(* CoDeSys 2.3.9.45 project: FillingStation.pro *)
(* Libraries: Standard.lib 2.12.10 14:48:34, SYSLIBCALLBACK.LIB 2.12.10 14:48:32 *)

(* PLC configuration (modules and I/O channels)
0753-0553 4 AO 0-20mA [Type_14_4_Channels] node 0, in %IB4 out %QB8 {INTTypePAAssignment = PLC; INTTypeModule = plugged}
  vwPumpPower AT %QW0 [WORDOnW_Q] Ch_1 Analog output
  AT %QW1 [WORDOnW_Q] Ch_2 Analog output
  AT %QW2 [WORDOnW_Q] Ch_3 Analog output
  AT %QW3 [WORDOnW_Q] Ch_4 Analog output
0750-0492 2 AI 4-20mA Diff Measurement Input [Type_8_2_Channels] node 1, in %IB4 out %QB8 {INTTypePAAssignment = PLC; INTTypeModule = plugged}
  vwRawPressure AT %IW0 [WORDOnW_I] Ch_1 Input word
  AT %IW1 [WORDOnW_I] Ch_2 Input word
0750-1515 8 DO 24V DC 0.5A/ 2-wire [Type_10_8_Channels] node 2, in %IB12 out %QB8 {INTTypePAAssignment = PLC; INTTypeModule = plugged}
  vbOpenSamsonValve AT %QX4.0 [BOOLOnX_Q] Ch_1 Digital output
  vbCloseSamsonValve AT %QX4.1 [BOOLOnX_Q] Ch_2 Digital output
  vbOpenDrainValve AT %QX4.2 [BOOLOnX_Q] Ch_3 Digital output
  vbSwitchOnPump AT %QX4.3 [BOOLOnX_Q] Ch_4 Digital output
  AT %QX4.4 [BOOLOnX_Q] Ch_5 Digital output
  AT %QX4.5 [BOOLOnX_Q] Ch_6 Digital output
  AT %QX4.6 [BOOLOnX_Q] Ch_7 Digital output
  AT %QX4.7 [BOOLOnX_Q] Ch_8 Digital output
0750-0459 4 AI 0-10V DC s.e. [Type_8_4_Channels] node 3, in %IB4 out %QB16 {INTTypePAAssignment = PLC; INTTypeModule = plugged}
  vwRawValvePosition AT %IW2 [WORDOnW_I] Ch_1 Input word
  AT %IW3 [WORDOnW_I] Ch_2 Input word
  AT %IW4 [WORDOnW_I] Ch_3 Input word
  AT %IW5 [WORDOnW_I] Ch_4 Input word
Fieldbus variables [FB_VARS] node 1, in %IB0 out %QB0
Flag variables [FLAG_VARS] node 2, in %IB0 out %QB0
Modbus-Master [MB_MASTER] node 3, in %IB0 out %QB0
*)

(* Global variable list: Globale_Variablen *)
VAR_GLOBAL
	vrWaterLevel:REAL;
	vrgrWaterLevel:ARRAY[1..16] OF REAL;
	vrStandardGravity:REAL:=9.81;
	viDensityWater:INT:=1000;
	vrValvePosition:REAL;
	vrValvePositionPercentage:REAL;
	vrValvePositionDesired:REAL;
	viPumpPowerPercentage:INT;
	vbManualValveControl:BOOL:=TRUE;
	vbAutomaticValveControl:BOOL:=FALSE;
	vbPreviousValveControl:STRING:='MANUAL';
	vbPreviousSamsonValveDirection:STRING:='STOP';
	vbStopSamsonValve:BOOL:=TRUE;
END_VAR

(* POU PLC_PRG, FBD *)
PROGRAM PLC_PRG
VAR
END_VAR
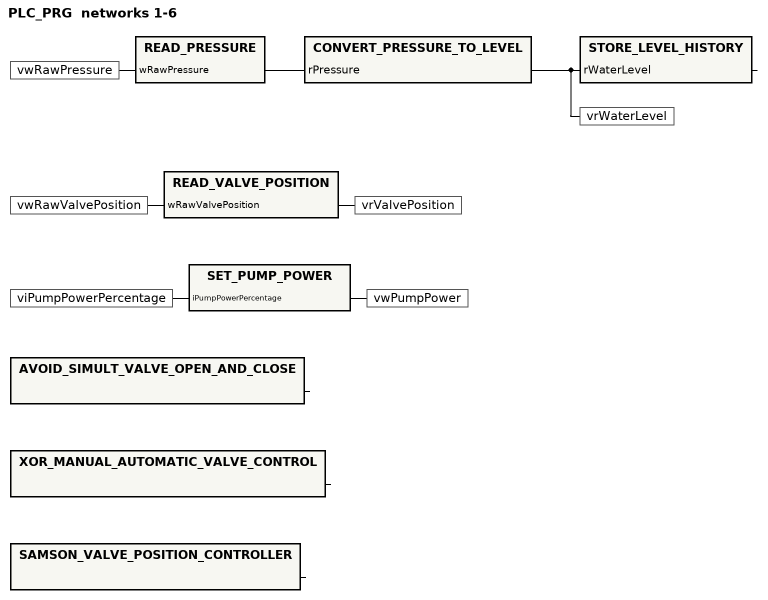
_FBD_ (* Function Block Diagram *)
NETWORK 1
	STORE_LEVEL_HISTORY(rWaterLevel: <CONVERT_PRESSURE_TO_LEVEL(rPressure: READ_PRESSURE(wRawPressure: vwRawPressure)) => vrWaterLevel>)
NETWORK 2
	READ_VALVE_POSITION(wRawValvePosition: vwRawValvePosition) => vrValvePosition
NETWORK 3
	SET_PUMP_POWER(iPumpPowerPercentage: viPumpPowerPercentage) => vwPumpPower
NETWORK 4
	AVOID_SIMULT_VALVE_OPEN_AND_CLOSE()
NETWORK 5
	XOR_MANUAL_AUTOMATIC_VALVE_CONTROL()
NETWORK 6
	SAMSON_VALVE_POSITION_CONTROLLER()
_END_FBD_
(* the same logic as Structured Text *)
(* Network 1: see the listing above *)
(* Network 2 *)
vrValvePosition := READ_VALVE_POSITION(wRawValvePosition := vwRawValvePosition);
(* Network 3 *)
vwPumpPower := SET_PUMP_POWER(iPumpPowerPercentage := viPumpPowerPercentage);
(* Network 4 *)
AVOID_SIMULT_VALVE_OPEN_AND_CLOSE();
(* Network 5 *)
XOR_MANUAL_AUTOMATIC_VALVE_CONTROL();
(* Network 6 *)
SAMSON_VALVE_POSITION_CONTROLLER();
END_PROGRAM

(* POU STORE_LEVEL_HISTORY, ST *)
FUNCTION STORE_LEVEL_HISTORY : BOOL
VAR_INPUT
	rWaterLevel:REAL;
END_VAR
VAR
	index: INT;
	rgrWaterLevelTmp:ARRAY[1..16] OF REAL;
	rgrWaterLevel: REAL;
END_VAR
rgrWaterLevelTmp := vrgrWaterLevel;

FOR index:=1 TO 15 DO
	vrgrWaterLevel[index]:= rgrWaterLevelTmp[index+1];
END_FOR

vrgrWaterLevel[16] := rWaterLevel;
END_FUNCTION

(* POU CONVERT_PRESSURE_TO_LEVEL, ST *)
FUNCTION CONVERT_PRESSURE_TO_LEVEL : REAL
VAR_INPUT
	rPressure:REAL;
END_VAR
VAR
END_VAR
CONVERT_PRESSURE_TO_LEVEL := rPressure/viDensityWater/vrStandardGravity;
END_FUNCTION

(* POU READ_PRESSURE, ST *)
FUNCTION READ_PRESSURE : REAL
VAR_INPUT
	wRawPressure:WORD;
END_VAR
VAR
END_VAR
READ_PRESSURE := WORD_TO_REAL(wRawPressure)/65535*100000;
END_FUNCTION

(* POU READ_VALVE_POSITION, ST *)
FUNCTION READ_VALVE_POSITION : REAL
VAR_INPUT
	wRawValvePosition:WORD;
END_VAR
VAR
END_VAR
READ_VALVE_POSITION := WORD_TO_REAL(wRawValvePosition)/65535*1;
vrValvePositionPercentage := READ_VALVE_POSITION*100;
END_FUNCTION

(* POU SET_PUMP_POWER, ST *)
FUNCTION SET_PUMP_POWER : WORD
VAR_INPUT
	iPumpPowerPercentage: INT;
END_VAR
VAR
END_VAR
SET_PUMP_POWER := INT_TO_WORD(iPumpPowerPercentage)*65535/100;
END_FUNCTION

(* POU AVOID_SIMULT_VALVE_OPEN_AND_CLOSE, ST *)
FUNCTION AVOID_SIMULT_VALVE_OPEN_AND_CLOSE : BOOL
VAR_INPUT
END_VAR
VAR
END_VAR
IF vbOpenSamsonValve AND vbStopSamsonValve THEN
	IF vbPreviousSamsonValveDirection = 'OPEN' THEN
		vbOpenSamsonValve := FALSE;
		vbStopSamsonValve := TRUE;
		vbCloseSamsonValve := FALSE;
		vbPreviousSamsonValveDirection := 'STOP';
	ELSIF vbPreviousSamsonValveDirection = 'STOP' THEN
		vbOpenSamsonValve := TRUE;
		vbStopSamsonValve := FALSE;
		vbCloseSamsonValve := FALSE;
		vbPreviousSamsonValveDirection := 'OPEN';
	END_IF
ELSIF vbStopSamsonValve AND vbCloseSamsonValve THEN
	IF vbPreviousSamsonValveDirection = 'STOP' THEN
		vbOpenSamsonValve := FALSE;
		vbStopSamsonValve := FALSE;
		vbCloseSamsonValve := TRUE;
		vbPreviousSamsonValveDirection := 'CLOSE';
	ELSIF vbPreviousSamsonValveDirection = 'CLOSE' THEN
		vbOpenSamsonValve := FALSE;
		vbStopSamsonValve := TRUE;
		vbCloseSamsonValve := FALSE;
		vbPreviousSamsonValveDirection := 'STOP';
	END_IF
ELSIF vbOpenSamsonValve AND vbCloseSamsonValve THEN
	IF vbPreviousSamsonValveDirection = 'OPEN' THEN
		vbOpenSamsonValve := FALSE;
		vbStopSamsonValve := FALSE;
		vbCloseSamsonValve := TRUE;
		vbPreviousSamsonValveDirection := 'CLOSE';
	ELSIF vbPreviousSamsonValveDirection = 'CLOSE' THEN
		vbOpenSamsonValve := TRUE;
		vbStopSamsonValve := FALSE;
		vbCloseSamsonValve := FALSE;
		vbPreviousSamsonValveDirection := 'OPEN';
	END_IF
END_IF

AVOID_SIMULT_VALVE_OPEN_AND_CLOSE := TRUE;
END_FUNCTION

(* POU XOR_MANUAL_AUTOMATIC_VALVE_CONTROL, ST *)
FUNCTION XOR_MANUAL_AUTOMATIC_VALVE_CONTROL : BOOL
VAR_INPUT
END_VAR
VAR
END_VAR
IF vbAutomaticValveControl AND vbManualValveControl THEN
	IF vbPreviousValveControl = 'MANUAL' THEN
			vbAutomaticValveControl := TRUE;
			vbManualValveControl := FALSE;
			vbPreviousValveControl := 'AUTOMATIC';
	ELSIF
			vbPreviousValveControl =  'AUTOMATIC' THEN
			vbAutomaticValveControl := FALSE;
			vbManualValveControl := TRUE;
			vbPreviousValveControl := 'MANUAL';
	END_IF
END_IF

XOR_MANUAL_AUTOMATIC_VALVE_CONTROL := TRUE;
END_FUNCTION

(* POU SAMSON_VALVE_POSITION_CONTROLLER, ST *)
FUNCTION SAMSON_VALVE_POSITION_CONTROLLER : BOOL
VAR_INPUT
END_VAR
VAR
	delta:REAL:=0.1;
END_VAR
IF vbAutomaticValveControl = TRUE THEN
	IF vrValvePosition < vrValvePositionDesired/100 - delta THEN
		vbOpenSamsonValve := TRUE;
		vbSTOPSamsonValve := FALSE;
		vbCloseSamsonValve := FALSE;
	ELSIF vrValvePosition > vrValvePositionDesired/100 + delta THEN
		vbOpenSamsonValve := FALSE;
		vbSTOPSamsonValve := FALSE;
		vbCloseSamsonValve := TRUE;
	END_IF
END_IF

SAMSON_VALVE_POSITION_CONTROLLER := TRUE;
END_FUNCTION

(* POU Configuration/MODBUS_CONFIGURATION, ST *)
PROGRAM MODBUS_CONFIGURATION        
VAR                                
END_VAR                            
(*                                 
   <?xml version="1.0" encoding="UTF-16" standalone="yes"?>
<network xml_structure_version="1" xml_feature_version="1">
	<generator_settings minRTUTaskCycleTimeMs="5" minEthaskCycleTimeMs="5" ethSlaveMultiplier="0.1" rtuInterfaceMultiplier="0.1" taskGeneration="false"/>
</network>
                              
*)                                 
;                                  
END_PROGRAM

(* Visualisation Filling_Station
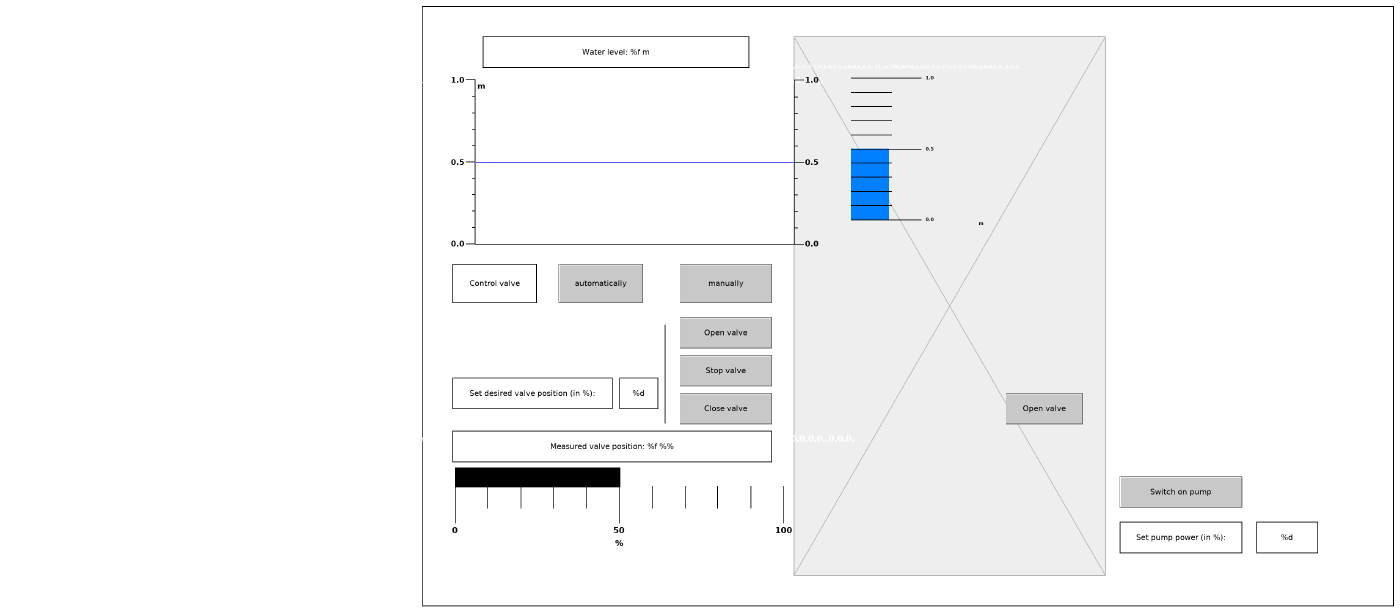
bitmap at (510,60)-(921,771): hydraulics-schematic-simplified.bmp
group at (510,100)-(931,311)
  rectangle at (0,0)-(1,1): text "{ExtendedElement},Visu\ElementDLL.ete,1,@Bargraph,211,421,2,1,0,vrWaterLevel,m,%.1f,0.1,0.5,0,1,0,0,0,0,0,0,0,-13,16,700,Arial,0,128,255,255,0,0,1,100,0,0,0,0,0,,0,0,0,"
  rectangle at (35,203)-(58,379): alarm colour if (vrWaterLevel) > 100; top ((vrWaterLevel * 1.0) - 0.5)  * -352
  rectangle at (80,368)-(196,389): text "0.0"
  rectangle at (80,193)-(196,214): text "0.5"
  rectangle at (80,17)-(196,38): text "1.0"
  rectangle at (103,380)-(127,396): text "m"
group at (60,110)-(541,341)
  rectangle at (0,8)-(1,9): text "{ExtendedElement},Visu\ElementDLL.ete,2,@Histogramm,481,231,vrgrWaterLevel,m,%.1f,0.1,0.5,0,1,0,0,0,0,0,0,0,-13,16,700,Arial,0,0,255,255,0,0,0,0,0,2,1,0_16,0,1,0,,"
  rectangle at (0,231)-(18,247): text "0.0"
  rectangle at (463,231)-(481,247): text "0.0"
  rectangle at (0,116)-(18,132): text "0.5"
  rectangle at (463,116)-(481,132): text "0.5"
  rectangle at (0,0)-(18,16): text "1.0"
  rectangle at (463,0)-(481,16): text "1.0"
  rectangle at (32,8)-(44,25): text "m"
  shape at (31,124)-(57,124): alarm colour if vrgrWaterLevel[0] < 0; top (-1.0 *  vrgrWaterLevel[1]  +  0.5  ) * 231 + SEL( vrgrWaterLevel[1] > 0.5 , 0.5, -0.5); bottom (-1.0 *  vrgrWaterLevel[0]  +  0.5  ) * 231 + SEL( vrgrWaterLevel[0] > 0.5 , 0.5, -0.5)
  shape at (57,124)-(83,124): alarm colour if vrgrWaterLevel[1] < 0; top (-1.0 *  vrgrWaterLevel[2]  +  0.5  ) * 231 + SEL( vrgrWaterLevel[2] > 0.5 , 0.5, -0.5); bottom (-1.0 *  vrgrWaterLevel[1]  +  0.5  ) * 231 + SEL( vrgrWaterLevel[1] > 0.5 , 0.5, -0.5)
  shape at (83,124)-(109,124): alarm colour if vrgrWaterLevel[2] < 0; top (-1.0 *  vrgrWaterLevel[3]  +  0.5  ) * 231 + SEL( vrgrWaterLevel[3] > 0.5 , 0.5, -0.5); bottom (-1.0 *  vrgrWaterLevel[2]  +  0.5  ) * 231 + SEL( vrgrWaterLevel[2] > 0.5 , 0.5, -0.5)
  shape at (109,124)-(135,124): alarm colour if vrgrWaterLevel[3] < 0; top (-1.0 *  vrgrWaterLevel[4]  +  0.5  ) * 231 + SEL( vrgrWaterLevel[4] > 0.5 , 0.5, -0.5); bottom (-1.0 *  vrgrWaterLevel[3]  +  0.5  ) * 231 + SEL( vrgrWaterLevel[3] > 0.5 , 0.5, -0.5)
  shape at (135,124)-(162,124): alarm colour if vrgrWaterLevel[4] < 0; top (-1.0 *  vrgrWaterLevel[5]  +  0.5  ) * 231 + SEL( vrgrWaterLevel[5] > 0.5 , 0.5, -0.5); bottom (-1.0 *  vrgrWaterLevel[4]  +  0.5  ) * 231 + SEL( vrgrWaterLevel[4] > 0.5 , 0.5, -0.5)
  shape at (162,124)-(188,124): alarm colour if vrgrWaterLevel[5] < 0; top (-1.0 *  vrgrWaterLevel[6]  +  0.5  ) * 231 + SEL( vrgrWaterLevel[6] > 0.5 , 0.5, -0.5); bottom (-1.0 *  vrgrWaterLevel[5]  +  0.5  ) * 231 + SEL( vrgrWaterLevel[5] > 0.5 , 0.5, -0.5)
  shape at (188,124)-(214,124): alarm colour if vrgrWaterLevel[6] < 0; top (-1.0 *  vrgrWaterLevel[7]  +  0.5  ) * 231 + SEL( vrgrWaterLevel[7] > 0.5 , 0.5, -0.5); bottom (-1.0 *  vrgrWaterLevel[6]  +  0.5  ) * 231 + SEL( vrgrWaterLevel[6] > 0.5 , 0.5, -0.5)
  shape at (214,124)-(240,124): alarm colour if vrgrWaterLevel[7] < 0; top (-1.0 *  vrgrWaterLevel[8]  +  0.5  ) * 231 + SEL( vrgrWaterLevel[8] > 0.5 , 0.5, -0.5); bottom (-1.0 *  vrgrWaterLevel[7]  +  0.5  ) * 231 + SEL( vrgrWaterLevel[7] > 0.5 , 0.5, -0.5)
  shape at (240,124)-(267,124): alarm colour if vrgrWaterLevel[8] < 0; top (-1.0 *  vrgrWaterLevel[9]  +  0.5  ) * 231 + SEL( vrgrWaterLevel[9] > 0.5 , 0.5, -0.5); bottom (-1.0 *  vrgrWaterLevel[8]  +  0.5  ) * 231 + SEL( vrgrWaterLevel[8] > 0.5 , 0.5, -0.5)
  shape at (267,124)-(293,124): alarm colour if vrgrWaterLevel[9] < 0; top (-1.0 *  vrgrWaterLevel[10]  +  0.5  ) * 231 + SEL( vrgrWaterLevel[10] > 0.5 , 0.5, -0.5); bottom (-1.0 *  vrgrWaterLevel[9]  +  0.5  ) * 231 + SEL( vrgrWaterLevel[9] > 0.5 , 0.5, -0.5)
  shape at (293,124)-(319,124): alarm colour if vrgrWaterLevel[10] < 0; top (-1.0 *  vrgrWaterLevel[11]  +  0.5  ) * 231 + SEL( vrgrWaterLevel[11] > 0.5 , 0.5, -0.5); bottom (-1.0 *  vrgrWaterLevel[10]  +  0.5  ) * 231 + SEL( vrgrWaterLevel[10] > 0.5 , 0.5, -0.5)
  shape at (319,124)-(345,124): alarm colour if vrgrWaterLevel[11] < 0; top (-1.0 *  vrgrWaterLevel[12]  +  0.5  ) * 231 + SEL( vrgrWaterLevel[12] > 0.5 , 0.5, -0.5); bottom (-1.0 *  vrgrWaterLevel[11]  +  0.5  ) * 231 + SEL( vrgrWaterLevel[11] > 0.5 , 0.5, -0.5)
  shape at (345,124)-(372,124): alarm colour if vrgrWaterLevel[12] < 0; top (-1.0 *  vrgrWaterLevel[13]  +  0.5  ) * 231 + SEL( vrgrWaterLevel[13] > 0.5 , 0.5, -0.5); bottom (-1.0 *  vrgrWaterLevel[12]  +  0.5  ) * 231 + SEL( vrgrWaterLevel[12] > 0.5 , 0.5, -0.5)
  shape at (372,124)-(398,124): alarm colour if vrgrWaterLevel[13] < 0; top (-1.0 *  vrgrWaterLevel[14]  +  0.5  ) * 231 + SEL( vrgrWaterLevel[14] > 0.5 , 0.5, -0.5); bottom (-1.0 *  vrgrWaterLevel[13]  +  0.5  ) * 231 + SEL( vrgrWaterLevel[13] > 0.5 , 0.5, -0.5)
  shape at (398,124)-(424,124): alarm colour if vrgrWaterLevel[14] < 0; top (-1.0 *  vrgrWaterLevel[15]  +  0.5  ) * 231 + SEL( vrgrWaterLevel[15] > 0.5 , 0.5, -0.5); bottom (-1.0 *  vrgrWaterLevel[14]  +  0.5  ) * 231 + SEL( vrgrWaterLevel[14] > 0.5 , 0.5, -0.5)
  shape at (424,124)-(450,124): alarm colour if vrgrWaterLevel[15] < 0; top (-1.0 *  vrgrWaterLevel[16]  +  0.5  ) * 231 + SEL( vrgrWaterLevel[16] > 0.5 , 0.5, -0.5); bottom (-1.0 *  vrgrWaterLevel[15]  +  0.5  ) * 231 + SEL( vrgrWaterLevel[15] > 0.5 , 0.5, -0.5)
group at (30,590)-(511,811)
  rectangle at (0,0)-(1,1): text "{ExtendedElement},Visu\ElementDLL.ete,1,@Bargraph,481,221,0,0,0,vrValvePositionPercentage,%,%.0f,10,50,0,100,0,0,0,0,0,0,0,-13,16,700,Arial,0,0,0,255,0,0,0,0,0,0,0,0,0,,0,0,0,"
  rectangle at (32,36)-(241,60): alarm colour if (vrValvePositionPercentage) < 0; right ((vrValvePositionPercentage * 1.0) - 50)  * 4.16
  rectangle at (27,106)-(36,206): text "0"
  rectangle at (230,106)-(249,206): text "50"
  rectangle at (434,106)-(462,206): text "100"
  rectangle at (230,121)-(250,137): text "%"
button at (790,530)-(891,571): text "Open valve"; toggles vbOpenDrainValve
button at (940,640)-(1101,681): text "Switch on pump"; toggles vbSwitchOnPump
rectangle at (100,60)-(451,101): text "Water level: %f m"; shows vrWaterLevel
rectangle at (60,580)-(481,621): text "Measured valve position: %f %%"; shows vrValvePositionPercentage
rectangle at (1120,700)-(1201,741): text "%d"; shows viPumpPowerPercentage; editable
rectangle at (940,700)-(1101,741): text "Set pump power (in %):"
button at (360,430)-(481,471): text "Open valve"; toggles vbOpenSamsonValve
button at (360,530)-(481,571): text "Close valve"; toggles vbCloseSamsonValve
rectangle at (60,360)-(171,411): text "Control valve"
button at (200,360)-(311,411): text "automatically"; toggles vbAutomaticValveControl
button at (360,360)-(481,411): text "manually"; toggles vbManualValveControl
rectangle at (60,510)-(271,551): text "Set desired valve position (in %):"
rectangle at (280,510)-(331,551): text "%d"; shows vrValvePositionDesired; editable
button at (360,480)-(481,521): text "Stop valve"; toggles vbStopSamsonValve
49 more shapes without text or variables
*)
